(* PLC project Untitled1, Beckhoff Automation GmbH TwinCAT PLC Control 3.5.13.20 *)
(* stored: creationDateTime 2020-07-06T12:35:27.715242, modificationDateTime 2020-07-06T12:35:27.715242 *)

PROGRAM MAIN
VAR
END_VAR

                  
                
END_PROGRAM

PROGRAM Example

VAR
	B: BOOL;
END_VAR

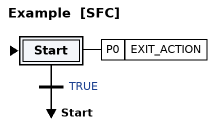
INITIAL_STEP Start:
  EXIT_ACTION(P0);
END_STEP
TRANSITION FROM Start TO Start
  := TRUE;
END_TRANSITION

ACTION EXIT_ACTION:
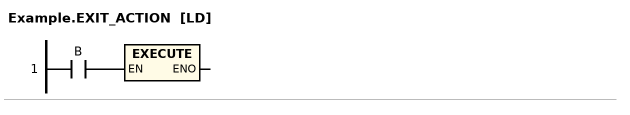
(* LD diagram, written out as Structured Text *)

IF B THEN
  B := FALSE;
END_IF;
END_ACTION
END_PROGRAM

CONFIGURATION Application
  RESOURCE Untitled1 ON PLC
    TASK PlcTask(INTERVAL := T#0ms, PRIORITY := 20);
    PROGRAM MAIN WITH PlcTask : MAIN;
  END_RESOURCE
END_CONFIGURATION
